PROGRAM pouStation6
VAR
	stationMode: FB_Mode;
	tCalcNumberOfPages: REAL;
	ceil: REAL;
	PartBuild: FB_PartBuild;
	retvall: UDINT;
	// TODO
	tPartPresent: BOOL;
END_VAR

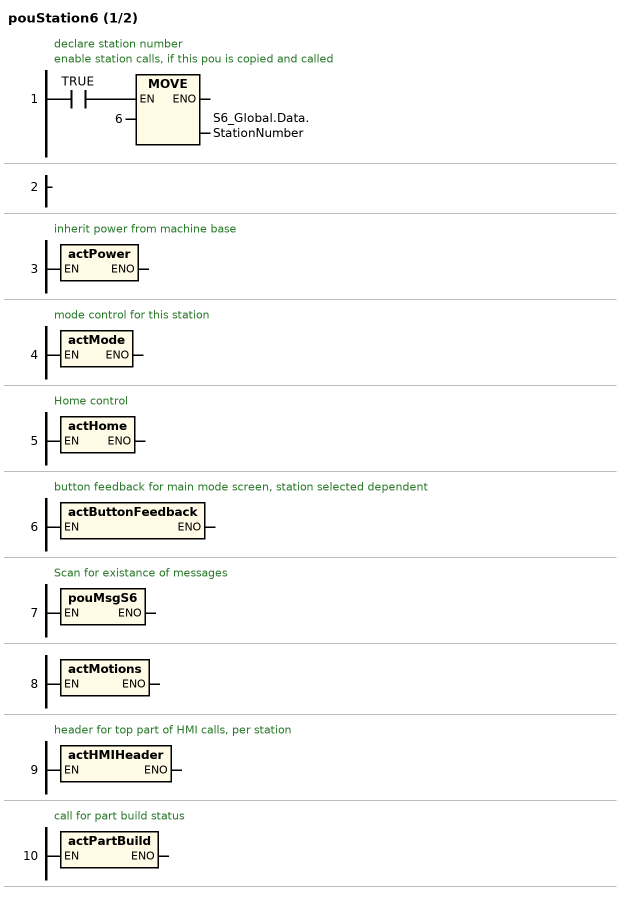
// NETWORK 1
// declare station number
// enable station calls, if this pou is copied and called
S6_Global.Data.StationNumber := 6;

// NETWORK 2

// NETWORK 3
// inherit power from machine base
actPower();

// NETWORK 4
// mode control for this station
actMode();

// NETWORK 5
// Home control
actHome();

// NETWORK 6
// button feedback for main mode screen, station selected dependent
actButtonFeedback();

// NETWORK 7
// Scan for existance of messages
pouMsgS6();

// NETWORK 8
actMotions();

// NETWORK 9
// header for top part of HMI calls, per station
actHMIHeader();

// NETWORK 10
// call for part build status
actPartBuild();

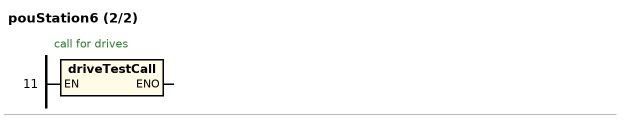
// NETWORK 11
// call for drives
driveTestCall();

ACTION actButtonFeedback:
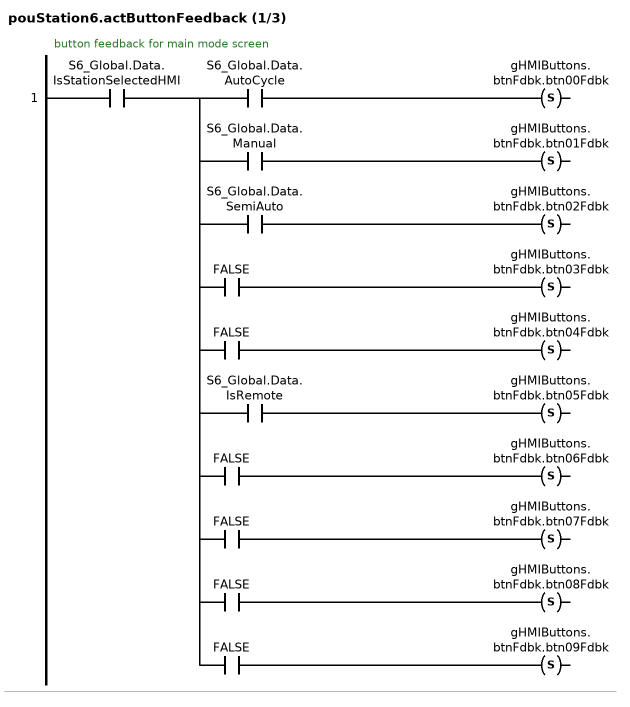
// NETWORK 1
// button feedback for main mode screen
gHMIButtons.btnFdbk.btn00Fdbk S= S6_Global.Data.IsStationSelectedHMI AND S6_Global.Data.AutoCycle;
gHMIButtons.btnFdbk.btn01Fdbk S= S6_Global.Data.IsStationSelectedHMI AND S6_Global.Data.Manual;
gHMIButtons.btnFdbk.btn02Fdbk S= S6_Global.Data.IsStationSelectedHMI AND S6_Global.Data.SemiAuto;
gHMIButtons.btnFdbk.btn03Fdbk S= S6_Global.Data.IsStationSelectedHMI AND FALSE;
gHMIButtons.btnFdbk.btn04Fdbk S= S6_Global.Data.IsStationSelectedHMI AND FALSE;
gHMIButtons.btnFdbk.btn05Fdbk S= S6_Global.Data.IsStationSelectedHMI AND S6_Global.Data.IsRemote;
gHMIButtons.btnFdbk.btn06Fdbk S= S6_Global.Data.IsStationSelectedHMI AND FALSE;
gHMIButtons.btnFdbk.btn07Fdbk S= S6_Global.Data.IsStationSelectedHMI AND FALSE;
gHMIButtons.btnFdbk.btn08Fdbk S= S6_Global.Data.IsStationSelectedHMI AND FALSE;
gHMIButtons.btnFdbk.btn09Fdbk S= S6_Global.Data.IsStationSelectedHMI AND FALSE;

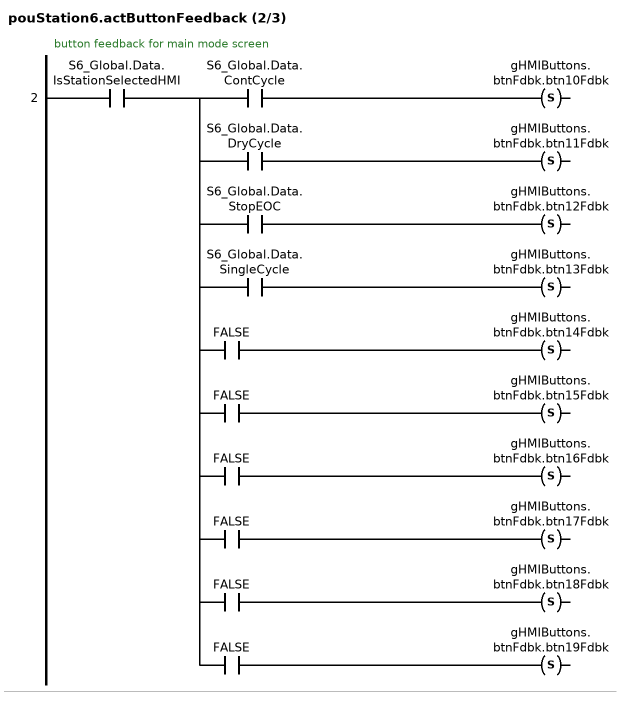
// NETWORK 2
// button feedback for main mode screen
gHMIButtons.btnFdbk.btn10Fdbk S= S6_Global.Data.IsStationSelectedHMI AND S6_Global.Data.ContCycle;
gHMIButtons.btnFdbk.btn11Fdbk S= S6_Global.Data.IsStationSelectedHMI AND S6_Global.Data.DryCycle;
gHMIButtons.btnFdbk.btn12Fdbk S= S6_Global.Data.IsStationSelectedHMI AND S6_Global.Data.StopEOC;
gHMIButtons.btnFdbk.btn13Fdbk S= S6_Global.Data.IsStationSelectedHMI AND S6_Global.Data.SingleCycle;
gHMIButtons.btnFdbk.btn14Fdbk S= S6_Global.Data.IsStationSelectedHMI AND FALSE;
gHMIButtons.btnFdbk.btn15Fdbk S= S6_Global.Data.IsStationSelectedHMI AND FALSE;
gHMIButtons.btnFdbk.btn16Fdbk S= S6_Global.Data.IsStationSelectedHMI AND FALSE;
gHMIButtons.btnFdbk.btn17Fdbk S= S6_Global.Data.IsStationSelectedHMI AND FALSE;
gHMIButtons.btnFdbk.btn18Fdbk S= S6_Global.Data.IsStationSelectedHMI AND FALSE;
gHMIButtons.btnFdbk.btn19Fdbk S= S6_Global.Data.IsStationSelectedHMI AND FALSE;

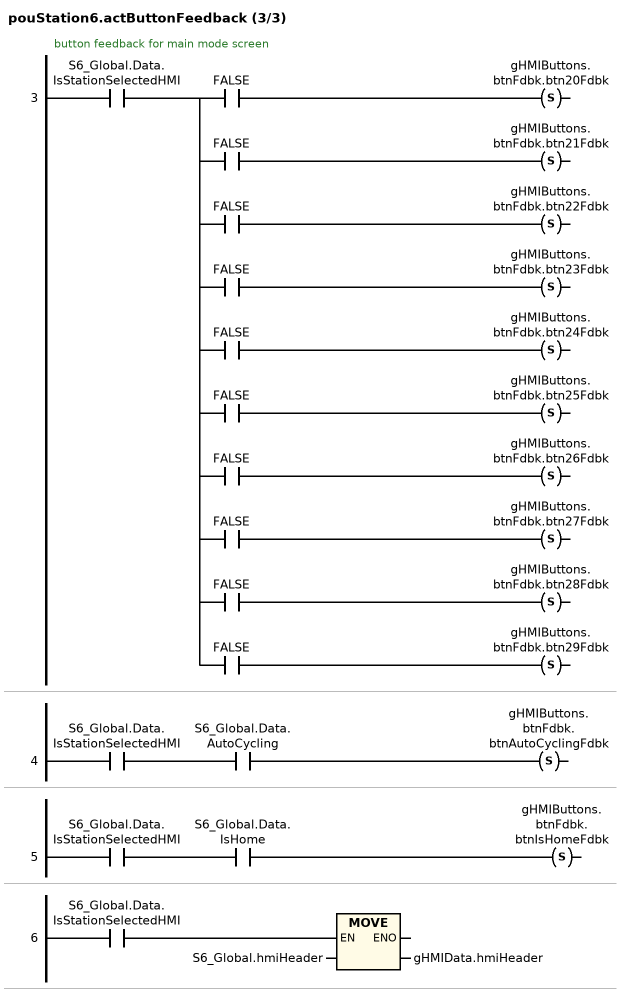
// NETWORK 3
// button feedback for main mode screen
gHMIButtons.btnFdbk.btn20Fdbk S= S6_Global.Data.IsStationSelectedHMI AND FALSE;
gHMIButtons.btnFdbk.btn21Fdbk S= S6_Global.Data.IsStationSelectedHMI AND FALSE;
gHMIButtons.btnFdbk.btn22Fdbk S= S6_Global.Data.IsStationSelectedHMI AND FALSE;
gHMIButtons.btnFdbk.btn23Fdbk S= S6_Global.Data.IsStationSelectedHMI AND FALSE;
gHMIButtons.btnFdbk.btn24Fdbk S= S6_Global.Data.IsStationSelectedHMI AND FALSE;
gHMIButtons.btnFdbk.btn25Fdbk S= S6_Global.Data.IsStationSelectedHMI AND FALSE;
gHMIButtons.btnFdbk.btn26Fdbk S= S6_Global.Data.IsStationSelectedHMI AND FALSE;
gHMIButtons.btnFdbk.btn27Fdbk S= S6_Global.Data.IsStationSelectedHMI AND FALSE;
gHMIButtons.btnFdbk.btn28Fdbk S= S6_Global.Data.IsStationSelectedHMI AND FALSE;
gHMIButtons.btnFdbk.btn29Fdbk S= S6_Global.Data.IsStationSelectedHMI AND FALSE;

// NETWORK 4
gHMIButtons.btnFdbk.btnAutoCyclingFdbk S= S6_Global.Data.IsStationSelectedHMI AND S6_Global.Data.AutoCycling;

// NETWORK 5
gHMIButtons.btnFdbk.btnIsHomeFdbk S= S6_Global.Data.IsStationSelectedHMI AND S6_Global.Data.IsHome;

// NETWORK 6
IF S6_Global.Data.IsStationSelectedHMI THEN gHMIData.hmiHeader := S6_Global.hmiHeader; END_IF
END_ACTION

ACTION actHMIHeader:
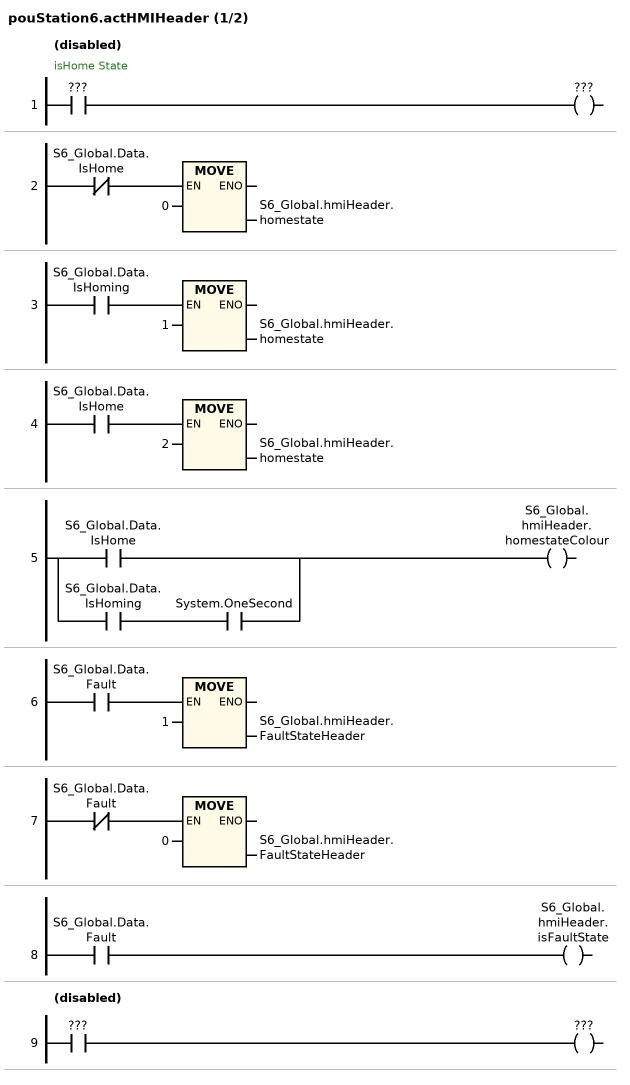
// NETWORK 1 (disabled)
// isHome State
// ??? := ???;

// NETWORK 2
IF NOT S6_Global.Data.IsHome THEN S6_Global.hmiHeader.homestate := 0; END_IF

// NETWORK 3
IF S6_Global.Data.IsHoming THEN S6_Global.hmiHeader.homestate := 1; END_IF

// NETWORK 4
IF S6_Global.Data.IsHome THEN S6_Global.hmiHeader.homestate := 2; END_IF

// NETWORK 5
S6_Global.hmiHeader.homestateColour := S6_Global.Data.IsHome OR S6_Global.Data.IsHoming AND System.OneSecond;

// NETWORK 6
IF S6_Global.Data.Fault THEN S6_Global.hmiHeader.FaultStateHeader := 1; END_IF

// NETWORK 7
IF NOT S6_Global.Data.Fault THEN S6_Global.hmiHeader.FaultStateHeader := 0; END_IF

// NETWORK 8
S6_Global.hmiHeader.isFaultState := S6_Global.Data.Fault;

// NETWORK 9 (disabled)
// ??? := ???;

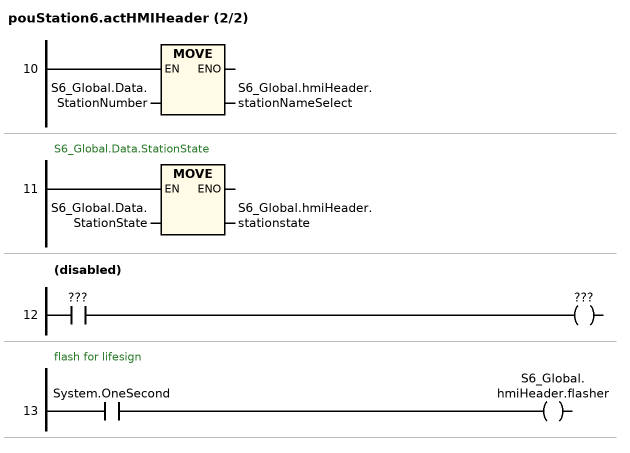
// NETWORK 10
S6_Global.hmiHeader.stationNameSelect := S6_Global.Data.StationNumber;

// NETWORK 11
// S6_Global.Data.StationState
S6_Global.hmiHeader.stationstate := S6_Global.Data.StationState;

// NETWORK 12 (disabled)
// ??? := ???;

// NETWORK 13
// flash for lifesign
S6_Global.hmiHeader.flasher := System.OneSecond;
END_ACTION

ACTION actHome:
//Set home status for station

IF 
//are all motions returned
S6_01_Motion_01_01.Motion.qReturnDepth AND
S6_01_Motion_01_02.Motion.qReturnDepth AND
S6_01_Motion_01_03.Motion.qReturnDepth AND
S6_01_Motion_01_04.Motion.qReturnDepth AND
S6_01_Motion_01_05.Motion.qReturnDepth AND
S6_01_Motion_01_06.Motion.qReturnDepth

	THEN
		//set IsHome value for station
		S6_Global.Data.IsHome := TRUE;
	ELSE
		S6_Global.Data.IsHome := FALSE;
END_IF
END_ACTION

ACTION actMaxNumStationPages:
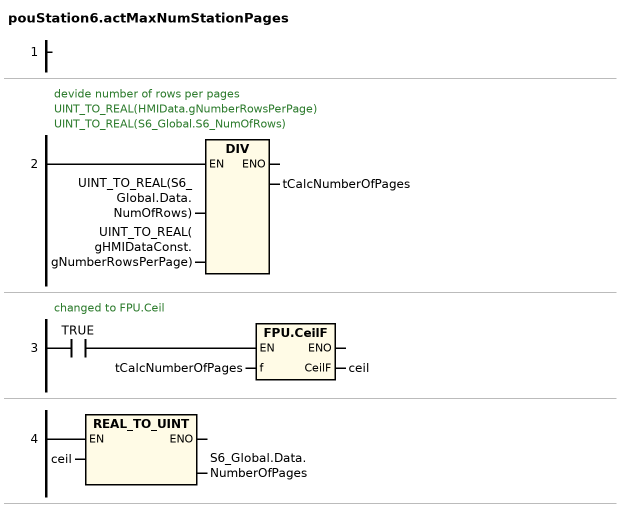
// NETWORK 1

// NETWORK 2
// devide number of rows per pages
// UINT_TO_REAL(HMIData.gNumberRowsPerPage)
// UINT_TO_REAL(S6_Global.S6_NumOfRows)
tCalcNumberOfPages := (UINT_TO_REAL(S6_Global.Data.NumOfRows)) / (UINT_TO_REAL(gHMIDataConst.gNumberRowsPerPage));

// NETWORK 3
// changed to FPU.Ceil
ceil := FPU.CeilF(f := tCalcNumberOfPages);

// NETWORK 4
S6_Global.Data.NumberOfPages := REAL_TO_UINT(ceil);
END_ACTION

ACTION actMode:
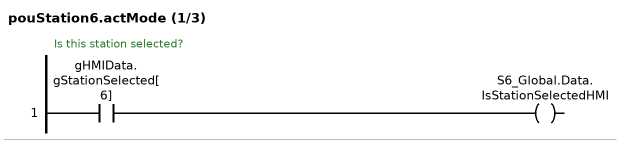
// NETWORK 1
// Is this station selected?
S6_Global.Data.IsStationSelectedHMI := gHMIData.gStationSelected[6];

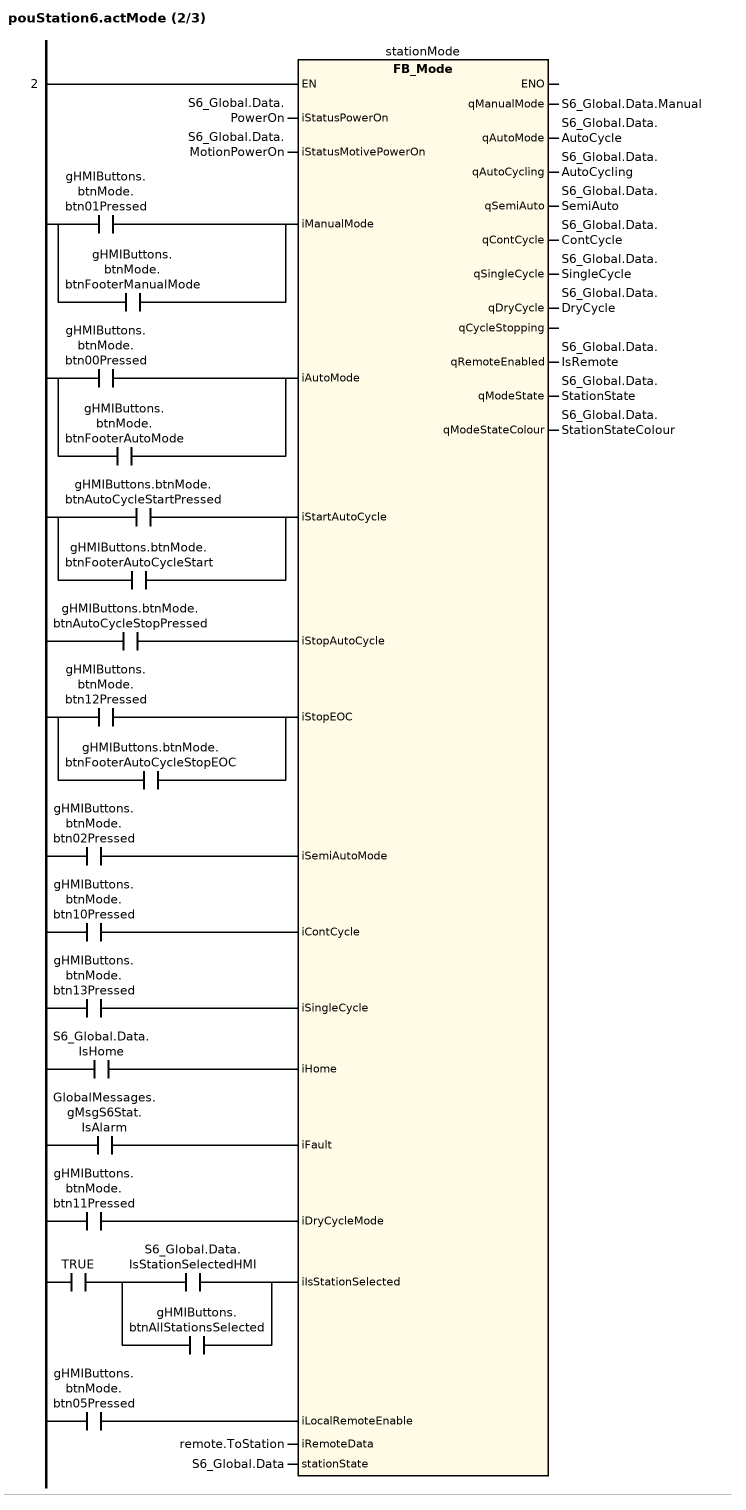
// NETWORK 2
stationMode(
    iStatusPowerOn := S6_Global.Data.PowerOn,
    iStatusMotivePowerOn := S6_Global.Data.MotionPowerOn,
    iManualMode := gHMIButtons.btnMode.btn01Pressed OR gHMIButtons.btnMode.btnFooterManualMode,
    iAutoMode := gHMIButtons.btnMode.btn00Pressed OR gHMIButtons.btnMode.btnFooterAutoMode,
    iStartAutoCycle := gHMIButtons.btnMode.btnAutoCycleStartPressed OR gHMIButtons.btnMode.btnFooterAutoCycleStart,
    iStopAutoCycle := gHMIButtons.btnMode.btnAutoCycleStopPressed,
    iStopEOC := gHMIButtons.btnMode.btn12Pressed OR gHMIButtons.btnMode.btnFooterAutoCycleStopEOC,
    iSemiAutoMode := gHMIButtons.btnMode.btn02Pressed,
    iContCycle := gHMIButtons.btnMode.btn10Pressed,
    iSingleCycle := gHMIButtons.btnMode.btn13Pressed,
    iHome := S6_Global.Data.IsHome,
    iFault := GlobalMessages.gMsgS6Stat.IsAlarm,
    iDryCycleMode := gHMIButtons.btnMode.btn11Pressed,
    iIsStationSelected := TRUE AND (S6_Global.Data.IsStationSelectedHMI OR gHMIButtons.btnAllStationsSelected),
    iLocalRemoteEnable := gHMIButtons.btnMode.btn05Pressed,
    iRemoteData := remote.ToStation,
    stationState := S6_Global.Data,
    qManualMode => S6_Global.Data.Manual,
    qAutoMode => S6_Global.Data.AutoCycle,
    qAutoCycling => S6_Global.Data.AutoCycling,
    qSemiAuto => S6_Global.Data.SemiAuto,
    qContCycle => S6_Global.Data.ContCycle,
    qSingleCycle => S6_Global.Data.SingleCycle,
    qDryCycle => S6_Global.Data.DryCycle,
    qRemoteEnabled => S6_Global.Data.IsRemote,
    qModeState => S6_Global.Data.StationState,
    qModeStateColour => S6_Global.Data.StationStateColour); // FB_Mode

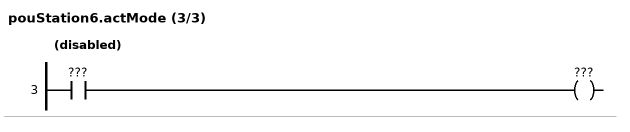
// NETWORK 3 (disabled)
// ??? := ???;
END_ACTION

ACTION actMotions:
//station 1 = 10000 index


//init number of rows
S6_Global.Data.NumOfRows := 0;

//page 1
S6_01_Motion_01_01();
S6_01_Motion_01_02();
S6_01_Motion_01_03();
S6_01_Motion_01_04();
S6_01_Motion_01_05();
S6_01_Motion_01_06();

//page 2
S6_01_Motion_02_07();
S6_01_Motion_02_08();
S6_01_Motion_02_09();
S6_01_Motion_02_10();
S6_01_Motion_02_11();
S6_01_Motion_02_12();

//page 3
S6_01_Motion_03_13();
S6_01_Motion_03_14();
S6_01_Motion_03_15();
S6_01_Motion_03_16();
S6_01_Motion_03_17();
S6_01_Motion_03_18();

//page 4
S6_01_Motion_04_19();
S6_01_Motion_04_20();
S6_01_Motion_04_21();
S6_01_Motion_04_22();
S6_01_Motion_04_23();
S6_01_Motion_04_24();

//page 5
S6_01_Motion_05_25();
S6_01_Motion_05_26();
S6_01_Motion_05_27();
S6_01_Motion_05_28();
S6_01_Motion_05_29();
S6_01_Motion_05_30();

//page 6
S6_01_Motion_06_31();
S6_01_Motion_06_32();
S6_01_Motion_06_33();
S6_01_Motion_06_34();
S6_01_Motion_06_35();
S6_01_Motion_06_36();

//must be called after motionRow calls
actMaxNumStationPages();
END_ACTION

ACTION actPartBuild:
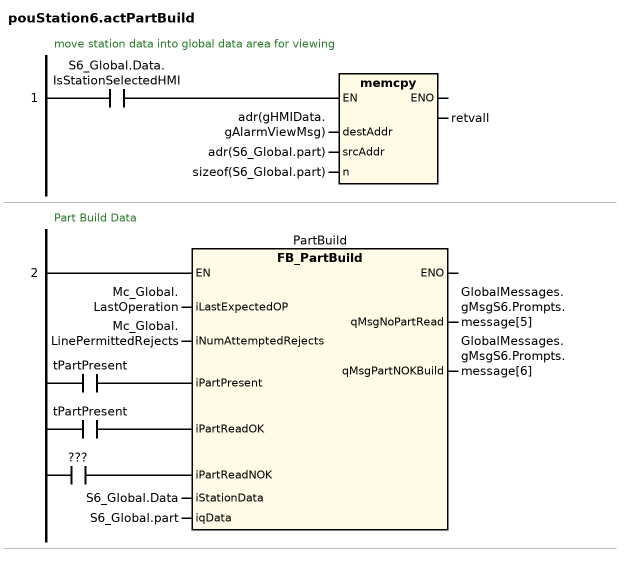
// NETWORK 1
// move station data into global data area for viewing
IF S6_Global.Data.IsStationSelectedHMI THEN
    retvall := memcpy(destAddr := adr(gHMIData.gAlarmViewMsg), srcAddr := adr(S6_Global.part), n := sizeof(S6_Global.part));
END_IF

// NETWORK 2
// Part Build Data
PartBuild(
    iLastExpectedOP := Mc_Global.LastOperation,
    iNumAttemptedRejects := Mc_Global.LinePermittedRejects,
    iPartPresent := tPartPresent,
    iPartReadOK := tPartPresent,
    iStationData := S6_Global.Data,
    iqData := S6_Global.part,
    qMsgNoPartRead => GlobalMessages.gMsgS6.Prompts.message[5],
    qMsgPartNOKBuild => GlobalMessages.gMsgS6.Prompts.message[6]); // FB_PartBuild
END_ACTION

ACTION actPower:
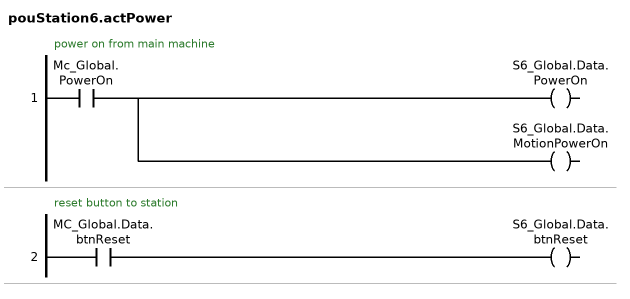
// NETWORK 1
// power on from main machine
S6_Global.Data.PowerOn := Mc_Global.PowerOn;
S6_Global.Data.MotionPowerOn := Mc_Global.PowerOn;

// NETWORK 2
// reset button to station
S6_Global.Data.btnReset := MC_Global.Data.btnReset;
END_ACTION

END_PROGRAM

(* stored: Version 1.1.0.1, ProductVersion 3.1.4024.12
   POU pouStation6: Id {218d0bcb-55ab-4645-b8b0-b412ea3cedea}, SpecialFunc None
   Action actButtonFeedback: Id {6f7b6a33-67df-4358-b64c-45fd776bf809}
   Action actHMIHeader: Id {60261169-f4e6-49e5-9632-a667087ff13e}
   Action actHome: Id {3ed5042f-aa22-48b5-a95b-2180ace66de5}
   Action actMaxNumStationPages: Id {9761c1f9-ecb1-422f-a1b5-4132970d06b0}
   Action actMode: Id {279d5167-9be0-4f6f-b83e-136df96b40ba}
   Action actMotions: Id {d189d6a7-1509-42ff-8964-dc104d37668a}
   Action actPartBuild: Id {01ba7381-2dff-4bf2-9b88-c7bc2e048c32}
   Action actPower: Id {0e81c3dd-6a6b-4648-aaad-10e3e93ab34d} *)
